INTERFACE I_FieldCodec

METHOD IsPackedRepeatedField : BOOL
VAR_INPUT
    nTag : UDINT;
END_VAR
END_METHOD

METHOD ValueReader : HRESULT
VAR_IN_OUT CONSTANT
    aBuffer : ARRAY [*] OF BYTE;   
END_VAR
VAR_IN_OUT
    stState : ST_ParserInternalState;
END_VAR
VAR_OUTPUT
    anyOut : T_Any;
END_VAR
END_METHOD

END_INTERFACE

(* stored: Version 1.1.0.1
   Itf I_FieldCodec: Id {efc0c207-4188-492e-bbf4-676d0a4c0d3b}
   Method IsPackedRepeatedField: Id {d897caca-16d3-4594-8894-ca03ec47971f}
   Method ValueReader: Id {3b7eefb9-456c-4f6e-87f8-51b5178c58ba} *)
